TYPE "Positioning_MOL_Machine_DataOut"
VERSION : 0.1
// Block: Positioning_MOL_Machine_DataOut
   STRUCT
      M_Contactor_Minus : Bool;
      M_Contactor_Plus : Bool;
   END_STRUCT;

END_TYPE
